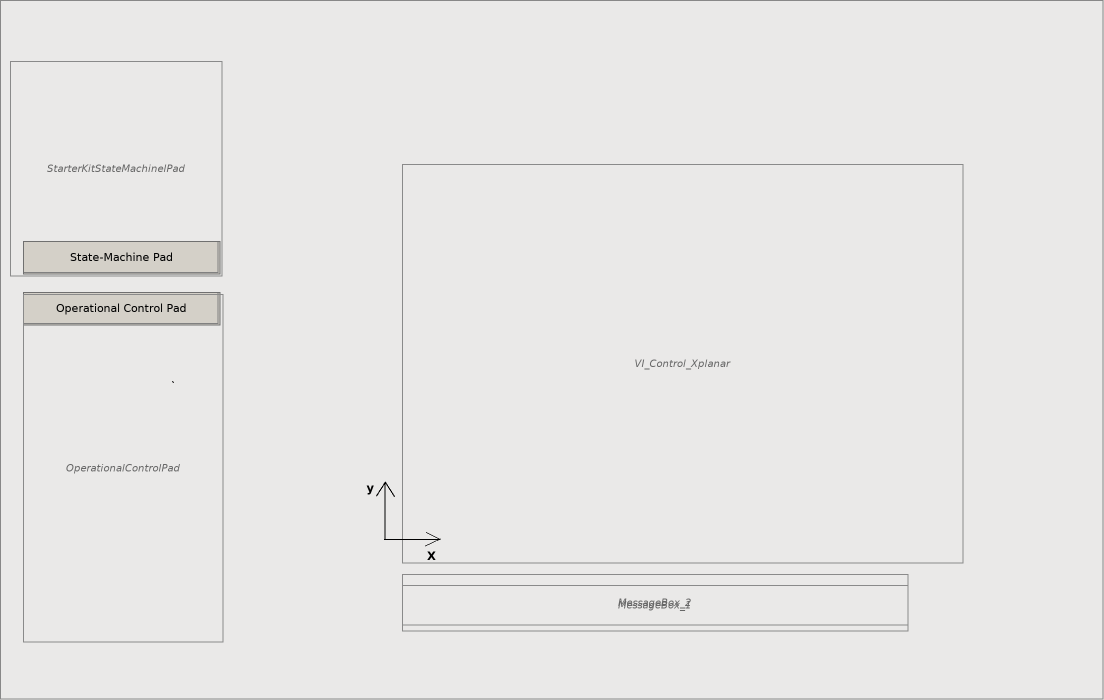
VISUALIZATION VI_MainSide  // 1104x700
    Polygon (172,381) (173,382)
    Frame (402,164 561x399)
        shows VI_Control_Xplanar()
    Button (23,292 197x33), "Operational Control Pad", invisible if: NOT stVisControl.stOperatorPad.bVisInvisible
        p3560616238: stVisControl.stOperatorPad.nButtonPositionX
        p2738717112: stVisControl.stOperatorPad.nButtonPositionY
        OnMouseClick: execute { stVisControl.stOperatorPad.bVisInvisibleButton := FALSE; }
    Button (23,241 197x33), "State-Machine Pad", invisible if: NOT stVisControl.stControlPad.bVisInvisible
        p3560616238: stVisControl.stControlPad.nButtonPositionX
        p2738717112: stVisControl.stControlPad.nButtonPositionY
        OnMouseClick: execute { stVisControl.stControlPad.bVisInvisibleButton := FALSE; }
    Frame (10,61 212x215), invisible if: stVisControl.stControlPad.bVisInvisible
        shows StarterKitStateMachinelPad(stControlPadControl := stVisControl.stControlPad)
        p3560616238: stVisControl.stControlPad.nFramePositionX
        p2738717112: stVisControl.stControlPad.nFramePositionY
    Frame (23,294 200x348), invisible if: stVisControl.stOperatorPad.bVisInvisible
        shows OperationalControlPad(stVisOperationalControl := stVisControl.stOperatorPad)
        p3560616238: stVisControl.stOperatorPad.nFramePositionX
        p2738717112: stVisControl.stOperatorPad.nFramePositionY
    Rectangle (1025,637 79x63)
    Group (357,473 88x98)
        Label (61,68 27x30), "X"
        Label (0,0 27x30), "y"
        Group (19,9 64x64)
            Line (8,57) (64,57)
            Line (50,50) (64,57)
            Line (64,57) (49,64)
            Line (9,57) (9,1)
            Line (9,0) (18,14)
            Line (9,0) (0,14)
    Frame (402,574 506x57), invisible if: NOT g_VisuMessage.bVisible_Box1_B
        shows MessageBox_2(message_1 := g_VisuMessage.sMessage_L1_Box1, message_2 := g_VisuMessage.sMessage_L2_Box1)
        tap g_VisuMessage.bAcknowledge
    Frame (402,585 506x40), invisible if: NOT g_VisuMessage.bVisible_Box1_A
        shows MessageBox_1(message_1 := g_VisuMessage.sMessage_L1_Box1)
END_VISUALIZATION

(* stored: Version 1.1.0.1
   Visu VI_MainSide: Id {676456b2-4c4e-43ae-9e93-f81d6d2ad0c3} *)
